{attribute 'GeneratedUsingTerminal: EP7402-0057-0017'}
{attribute addProperty BoxType "EP7402-0057-0017"}
{attribute addProperty Id "Device_DiagAT %I*Device_Diag_1464ECF921"}
{attribute addProperty CRC "2753397846"}
{attribute addProperty Size "21"}
TYPE STM_Inputs_Device_A41D8456 :
STRUCT
	{attribute addProperty Name "Device_Diag"}
	Device_Diag AT %I* : Device_Diag_1464ECF9;
END_STRUCT
END_TYPE

(* stored: Version 1.2.0.0, ProductVersion 3.1.4024.9
   DUT STM_Inputs_Device_A41D8456: Id {d4a5abbd-e0b5-4806-a628-7717538b02fa} *)
